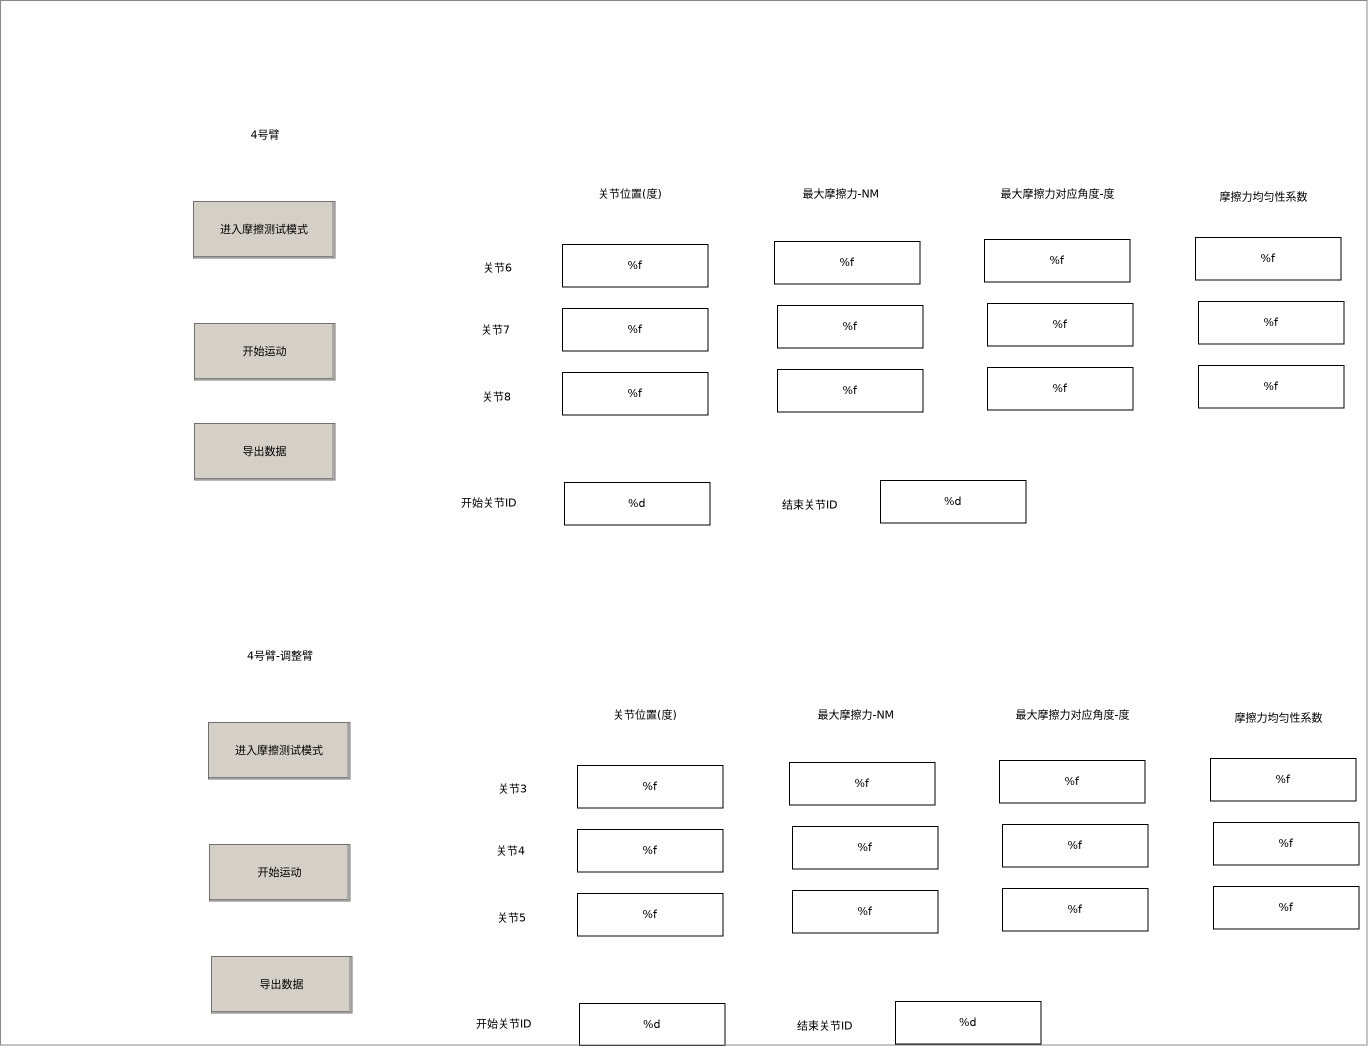
VISUALIZATION friction_a4  // 1368x1046
    Button (193,201 142x57), "进入摩擦测试模式", colour toggle: g_frictionTest.m_testMode[4]
        toggle g_frictionTest.m_testMode[4]
    Button (194,323 141x57), "开始运动", colour toggle: g_frictionTest.m_startMotion[4]
        toggle g_frictionTest.m_startMotion[4]
    Label (190,120 150x30), "4号臂"
    Rectangle (774,241 146x43), "%f", text variable: g_frictionTest.m_CoulombFrictionMax[4][1]
    Rectangle (777,305 146x43), "%f", text variable: g_frictionTest.m_CoulombFrictionMax[4][2]
    Rectangle (777,369 146x43), "%f", text variable: g_frictionTest.m_CoulombFrictionMax[4][3]
    Label (766,179 150x30), "最大摩擦力-NM"
    Rectangle (984,239 146x43), "%f", text variable: g_frictionTest.m_CoulombFrictionMax_JntPos[4][1]
    Rectangle (987,303 146x43), "%f", text variable: g_frictionTest.m_CoulombFrictionMax_JntPos[4][2]
    Rectangle (987,367 146x43), "%f", text variable: g_frictionTest.m_CoulombFrictionMax_JntPos[4][3]
    Label (941,179 233x30), "最大摩擦力对应角度-度"
    Rectangle (1195,237 146x43), "%f", text variable: g_frictionTest.m_CoulombFrictionRatio[4,1]
    Rectangle (1198,301 146x43), "%f", text variable: g_frictionTest.m_CoulombFrictionRatio[4,2]
    Rectangle (1198,365 146x43), "%f", text variable: g_frictionTest.m_CoulombFrictionRatio[4,3]
    Label (1174,182 179x30), "摩擦力均匀性系数"
    Rectangle (562,244 146x43), "%f", text variable: g_frictionTest.m_armDHJntPos[4][1]
    Label (446,250 103x36), "关节6"
    Label (444,312 103x36), "关节7"
    Label (445,379 103x36), "关节8"
    Rectangle (562,308 146x43), "%f", text variable: g_frictionTest.m_armDHJntPos[4][2]
    Rectangle (562,372 146x43), "%f", text variable: g_frictionTest.m_armDHJntPos[4][3]
    Label (555,179 150x30), "关节位置(度)"
    Label (414,488 150x30), "开始关节ID"
    Rectangle (564,482 146x43), "%d", text variable: g_frictionTest.m_jntIdStart[4]
        OnMouseClick: write the text variable via Default
    Label (735,490 150x30), "结束关节ID"
    Rectangle (880,480 146x43), "%d", text variable: g_frictionTest.m_jntIdEnd[4]
        OnMouseClick: write the text variable via Default
    Button (208,722 142x57), "进入摩擦测试模式", colour toggle: g_frictionTestSetup.m_testMode[4]
        toggle g_frictionTestSetup.m_testMode[4]
    Button (209,844 141x57), "开始运动", colour toggle: g_frictionTestSetup.m_startMotion[4]
        toggle g_frictionTestSetup.m_startMotion[4] p2164770859=TRUE
    Label (205,641 150x30), "4号臂-调整臂"
    Rectangle (789,762 146x43), "%f", text variable: g_frictionTestSetup.m_CoulombFrictionMax[4][3]
    Rectangle (792,826 146x43), "%f", text variable: g_frictionTestSetup.m_CoulombFrictionMax[4][4]
    Rectangle (792,890 146x43), "%f", text variable: g_frictionTestSetup.m_CoulombFrictionMax[4][5]
    Label (781,700 150x30), "最大摩擦力-NM"
    Rectangle (999,760 146x43), "%f", text variable: g_frictionTestSetup.m_CoulombFrictionMax_JntPos[4][3]
    Rectangle (1002,824 146x43), "%f", text variable: g_frictionTestSetup.m_CoulombFrictionMax_JntPos[4][4]
    Rectangle (1002,888 146x43), "%f", text variable: g_frictionTestSetup.m_CoulombFrictionMax_JntPos[4][5]
    Label (956,700 233x30), "最大摩擦力对应角度-度"
    Rectangle (1210,758 146x43), "%f", text variable: g_frictionTestSetup.m_CoulombFrictionRatio[4,3]
    Rectangle (1213,822 146x43), "%f", text variable: g_frictionTestSetup.m_CoulombFrictionRatio[4,4]
    Rectangle (1213,886 146x43), "%f", text variable: g_frictionTestSetup.m_CoulombFrictionRatio[4,5]
    Label (1189,703 179x30), "摩擦力均匀性系数"
    Rectangle (577,765 146x43), "%f", text variable: g_frictionTestSetup.m_armDHJntPos[4][3]
    Label (461,771 103x36), "关节3"
    Label (459,833 103x36), "关节4"
    Label (460,900 103x36), "关节5"
    Rectangle (577,829 146x43), "%f", text variable: g_frictionTestSetup.m_armDHJntPos[4][4]
    Rectangle (577,893 146x43), "%f", text variable: g_frictionTestSetup.m_armDHJntPos[4][5]
    Label (570,700 150x30), "关节位置(度)"
    Label (429,1009 150x30), "开始关节ID"
    Rectangle (579,1003 146x43), "%d", text variable: g_frictionTestSetup.m_jntIdStart[4]
        OnMouseClick: write the text variable via Default
    Label (750,1011 150x30), "结束关节ID"
    Rectangle (895,1001 146x43), "%d", text variable: g_frictionTestSetup.m_jntIdEnd[4]
        OnMouseClick: write the text variable via Default
    Button (194,423 141x57), "导出数据", colour toggle: g_frictionTest.m_duringWriteData[4]
        tap g_frictionTest.m_writeData[4]
    Button (211,956 141x57), "导出数据", colour toggle: g_frictionTestSetup.m_duringWriteData[4]
        tap g_frictionTestSetup.m_writeData[4]
END_VISUALIZATION

(* stored: Version 1.1.0.1, ProductVersion 3.1.4024.12
   Visu friction_a4: Id {f2c87ca5-a2dc-4bad-b0f0-43f4bc036911} *)
